(* PLC project Tc2_Standard.CTU Demo, tc3-libraries-kb TwinCAT 3.1 *)
(* stored: creationDateTime 2026-05-10T08:00:00, modificationDateTime 2026-05-10T08:00:00 *)

PROGRAM P_Demo_CTU
  VAR
    fbCTU : CTU;  (* Counter 实例 *)
    bReset : BOOL;  (* 复位计数到 0 *)
    bCountUp : BOOL;  (* 每个产品到位给一次上升沿 *)
    bFull : BOOL;  (* 达到 10 件时 TRUE *)
    nCV : WORD;  (* 已累计件数（监视） *)
  END_VAR

            // ============================================================
// Tc2_Standard.CTU 演示程序
// ============================================================
// 场景：累计 10 个产品后发出'换托盘'信号
// 验证步骤：
//   1. 把本 PROGRAM 加到 PlcTask 调用列表
//   2. 编译并登录目标
//   1. 强制 bReset := TRUE 一个周期 → nCV 归 0、bFull = FALSE
//   2. 重复给 bCountUp 上升沿 10 次 → nCV 增到 10、bFull = TRUE
//   3. CV >= PV 后的进一步行为 PDF 未描述（⚠️ 待人工确认）
// ============================================================

fbCTU(
    CU    := bCountUp,
    RESET := bReset,
    PV    := WORD#10,
    Q     => bFull,
    CV    => nCV
);

          
END_PROGRAM
